// TIA Portal V21 export
FUNCTION "AiFc" : Void   // FC108, LAD
{ S7_Optimized_Access := 'TRUE' }
// stored: AutoNumber false, SetENOAutomatically false
BEGIN

REGION Network 1: "AiDb"
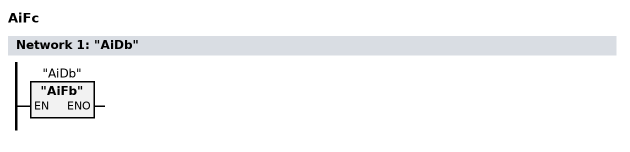
   RUNG wire#powerrail
      "AiDb"()
   END_RUNG
   // the same network as SCL:
   "AiDb"();   // "AiFb"
END_REGION

REGION Network 2 (SCL): AnalogInputIw
   "AiDb".Ai01.AnalogInputIw := "Ticr01NfcoLineTemp";
   "AiDb".Ai02.AnalogInputIw := "Ticr02VfcoLineTemp";
   "AiDb".Ai03.AnalogInputIw := "AiSpare01";
   "AiDb".Ai04.AnalogInputIw := "AiSpare02";
   "AiDb".Ai05.AnalogInputIw := "AiSpare03";
   "AiDb".Ai06.AnalogInputIw := "Ticr06Pf01InLineTemp";
   "AiDb".Ai07.AnalogInputIw := "Ticr07Pf02InLineTemp";
   "AiDb".Ai08.AnalogInputIw := "Ticr08Pf02OutLineTemp";
   "AiDb".Ai09.AnalogInputIw := "Ticr09PtlDrainTemp";
   "AiDb".Ai10.AnalogInputIw := "Ticr10VesselTemp";
   "AiDb".Ai11.AnalogInputIw := "Picr01VesselPressure";
   "AiDb".Ai12.AnalogInputIw := "Picr02VesselRclLine";
   "AiDb".Ai13.AnalogInputIw := "Picr03Pf01OutLinePressure";
   "AiDb".Ai14.AnalogInputIw := "Picr04Pf02OutLinePressure";
   "AiDb".Ai15.AnalogInputIw := "Cicr01ProcessDrainConductivity";
   "AiDb".Ai16.AnalogInputIw := "AiSpare04";
   "AiDb".Ai17.AnalogInputIw := "AiSpare05";
   "AiDb".Ai18.AnalogInputIw := "AiSpare06";
   "AiDb".Ai19.AnalogInputIw := "AiSpare07";
   "AiDb".Ai20.AnalogInputIw := "AiSpare08";
   "AiDb".Ai21.AnalogInputIw := "AiSpare09";
   "AiDb".Ai22.AnalogInputIw := "AiSpare10";
   "AiDb".Ai23.AnalogInputIw := "AiSpare11";
   "AiDb".Ai24.AnalogInputIw := "AiSpare12";
END_REGION
END_FUNCTION
